FUNCTION_BLOCK CMD_bloc (* Basic Function Block Type *)
  (* Standard: 61499-2 *)
  (* Version 0.0, 13/06/2022, Etienne, Schneider Electric, Template *)
  PACKAGE Main;
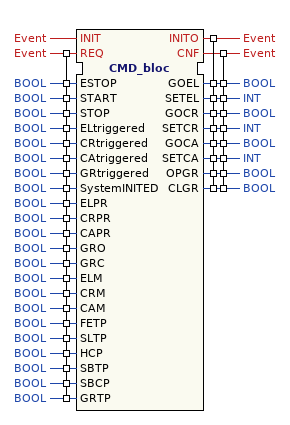
  EVENT_INPUT
    INIT; (* Initialization Request *)
    REQ WITH ESTOP, START, STOP, ELtriggered, CRtriggered, CAtriggered, GRtriggered, SystemINITED, ELPR, CRPR, CAPR, GRO, GRC, ELM, CRM, CAM, HCP, SBTP, SBCP, FETP, SLTP, GRTP; (* Normal Execution Request *)
  END_EVENT
  EVENT_OUTPUT
    INITO WITH GOEL, SETEL, GOCA, SETCA, GOCR, SETCR, OPGR, CLGR; (* Initialization Confirm *)
    CNF WITH GOEL, SETEL, GOCA, SETCA, GOCR, SETCR, OPGR, CLGR; (* Execution Confirmation *)
  END_EVENT
  VAR_INPUT
    ESTOP : BOOL;
    START : BOOL;
    STOP : BOOL;
    ELtriggered : BOOL;
    CRtriggered : BOOL;
    CAtriggered : BOOL;
    GRtriggered : BOOL;
    SystemINITED : BOOL;
    ELPR : BOOL;
    CRPR : BOOL;
    CAPR : BOOL;
    GRO : BOOL;
    GRC : BOOL;
    ELM : BOOL;
    CRM : BOOL;
    CAM : BOOL;
    FETP : BOOL;
    SLTP : BOOL;
    HCP : BOOL;
    SBTP : BOOL;
    SBCP : BOOL;
    GRTP : BOOL;
  END_VAR
  VAR_OUTPUT
    GOEL : BOOL; (* Output event qualifier *)
    SETEL : INT;
    GOCR : BOOL;
    SETCR : INT;
    GOCA : BOOL;
    SETCA : INT;
    OPGR : BOOL;
    CLGR : BOOL;
  END_VAR
  VAR
    i : INT;
  END_VAR
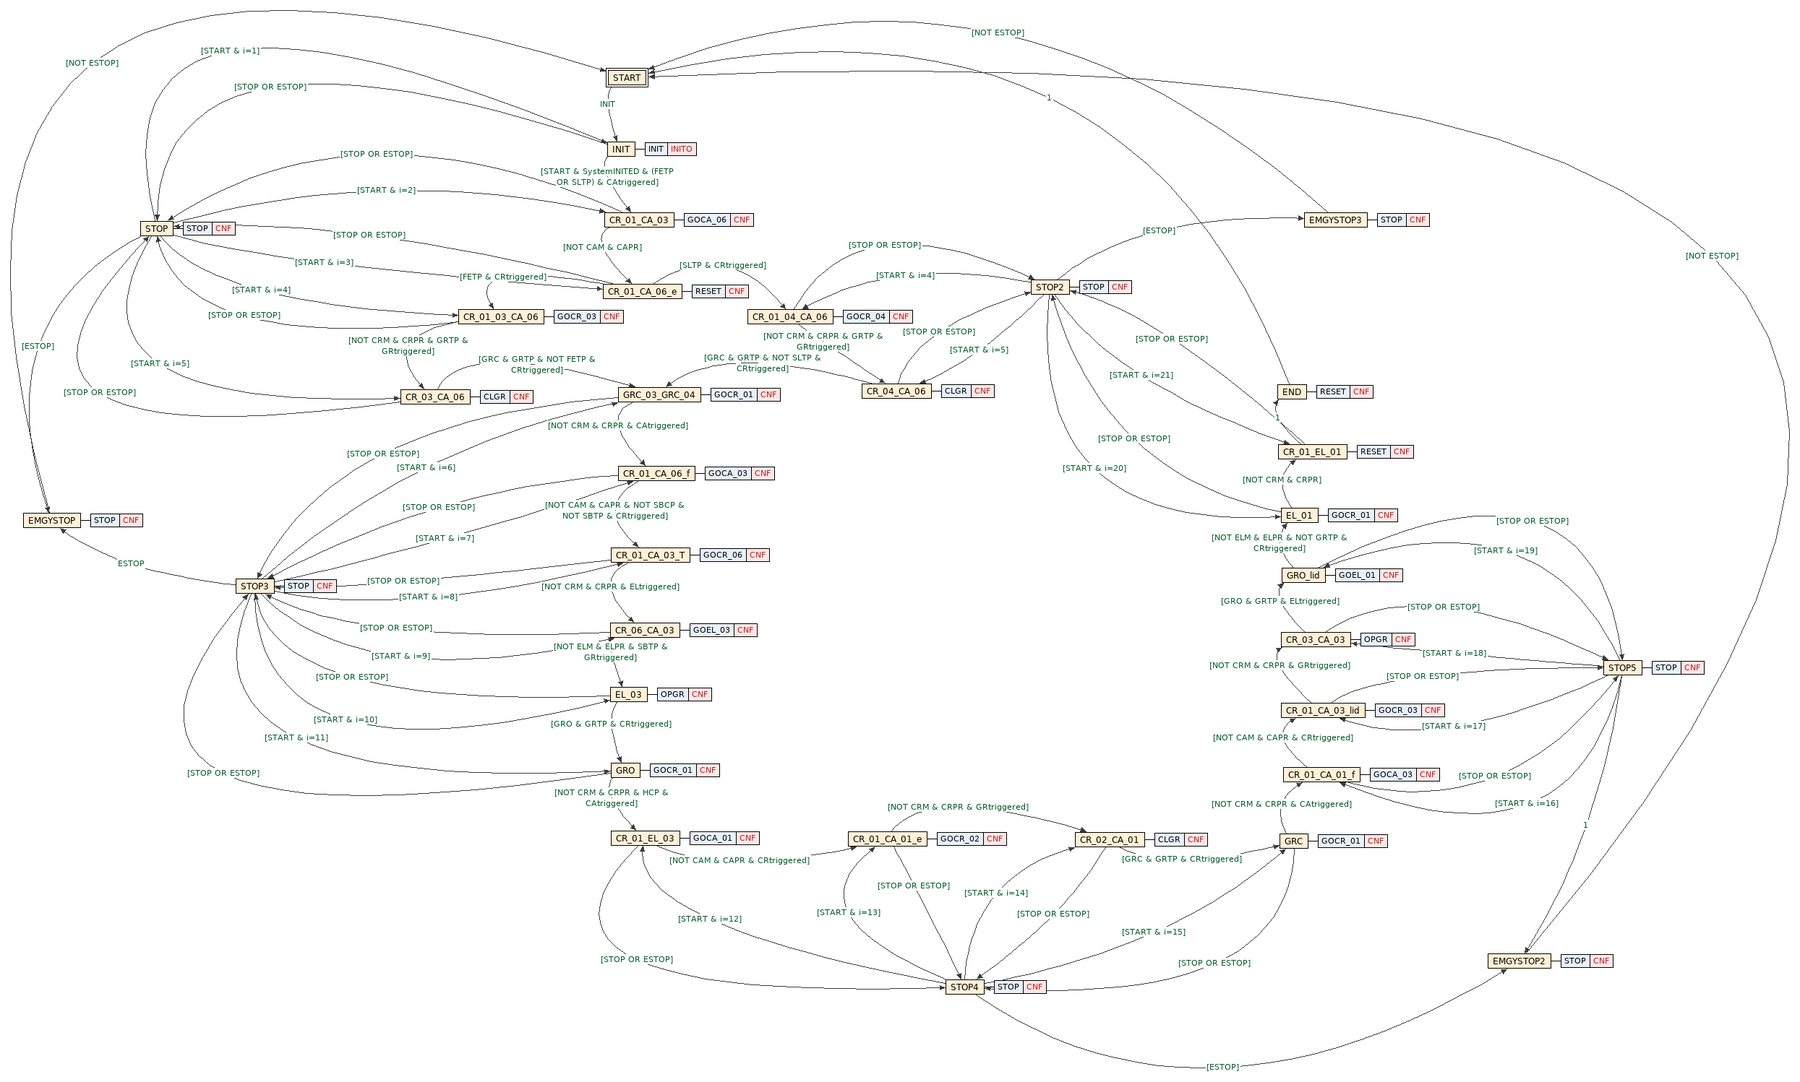
  EC_STATES
    START; (* Initial State *)
    INIT : INIT -> INITO; (* Initialization *)
    CR_01_CA_03 : GOCA_06 -> CNF;
    CR_01_03_CA_06 : GOCR_03 -> CNF;
    CR_01_04_CA_06 : GOCR_04 -> CNF;
    GRC_03_GRC_04 : GOCR_01 -> CNF;
    CR_01_CA_06_f : GOCA_03 -> CNF;
    CR_01_CA_03_T : GOCR_06 -> CNF;
    CR_06_CA_03 : GOEL_03 -> CNF;
    EL_03 : OPGR -> CNF;
    GRO : GOCR_01 -> CNF;
    EL_01 : GOCR_01 -> CNF;
    CR_01_EL_03 : GOCA_01 -> CNF;
    END : RESET -> CNF;
    CR_01_CA_01_e : GOCR_02 -> CNF;
    CR_02_CA_01 : CLGR -> CNF;
    GRC : GOCR_01 -> CNF;
    CR_01_CA_01_f : GOCA_03 -> CNF;
    CR_01_CA_03_lid : GOCR_03 -> CNF;
    CR_03_CA_03 : OPGR -> CNF;
    GRO_lid : GOEL_01 -> CNF;
    CR_01_EL_01 : RESET -> CNF;
    CR_01_CA_06_e : RESET -> CNF;
    CR_03_CA_06 : CLGR -> CNF;
    CR_04_CA_06 : CLGR -> CNF;
    STOP : STOP -> CNF;
    STOP2 : STOP -> CNF;
    STOP3 : STOP -> CNF;
    STOP4 : STOP -> CNF;
    STOP5 : STOP -> CNF;
    EMGYSTOP : STOP -> CNF;
    EMGYSTOP2 : STOP -> CNF;
    EMGYSTOP3 : STOP -> CNF;
  END_STATES
  EC_TRANSITIONS
    START TO INIT := INIT;
    CR_01_03_CA_06 TO CR_03_CA_06 := [NOT CRM & CRPR & GRTP & GRtriggered];
    CR_01_04_CA_06 TO CR_04_CA_06 := [NOT CRM & CRPR & GRTP & GRtriggered];
    GRC_03_GRC_04 TO CR_01_CA_06_f := [NOT CRM & CRPR & CAtriggered];
    CR_01_CA_06_f TO CR_01_CA_03_T := [NOT CAM & CAPR & NOT SBCP & NOT SBTP & CRtriggered];
    CR_01_CA_03_T TO CR_06_CA_03 := [NOT CRM & CRPR & ELtriggered];
    CR_06_CA_03 TO EL_03 := [NOT ELM & ELPR & SBTP & GRtriggered];
    EL_03 TO GRO := [GRO & GRTP & CRtriggered];
    GRO TO CR_01_EL_03 := [NOT CRM & CRPR & HCP & CAtriggered];
    CR_01_EL_03 TO CR_01_CA_01_e := [NOT CAM & CAPR & CRtriggered];
    CR_01_CA_01_e TO CR_02_CA_01 := [NOT CRM & CRPR & GRtriggered];
    CR_02_CA_01 TO GRC := [GRC & GRTP & CRtriggered];
    GRC TO CR_01_CA_01_f := [NOT CRM & CRPR & CAtriggered];
    CR_01_CA_01_f TO CR_01_CA_03_lid := [NOT CAM & CAPR & CRtriggered];
    CR_01_CA_03_lid TO CR_03_CA_03 := [NOT CRM & CRPR & GRtriggered];
    CR_03_CA_03 TO GRO_lid := [GRO & GRTP & ELtriggered];
    GRO_lid TO EL_01 := [NOT ELM & ELPR & NOT GRTP & CRtriggered];
    EL_01 TO CR_01_EL_01 := [NOT CRM & CRPR];
    END TO START := 1;
    CR_01_CA_03 TO CR_01_CA_06_e := [NOT CAM & CAPR];
    CR_01_CA_06_e TO CR_01_03_CA_06 := [FETP & CRtriggered];
    CR_01_CA_06_e TO CR_01_04_CA_06 := [SLTP & CRtriggered];
    CR_03_CA_06 TO GRC_03_GRC_04 := [GRC & GRTP & NOT FETP & CRtriggered];
    CR_04_CA_06 TO GRC_03_GRC_04 := [GRC & GRTP & NOT SLTP & CRtriggered];
    INIT TO STOP := [STOP OR ESTOP];
    CR_01_CA_03 TO STOP := [STOP OR ESTOP];
    CR_01_CA_06_e TO STOP := [STOP OR ESTOP];
    CR_01_03_CA_06 TO STOP := [STOP OR ESTOP];
    CR_03_CA_06 TO STOP := [STOP OR ESTOP];
    CR_01_04_CA_06 TO STOP2 := [STOP OR ESTOP];
    CR_04_CA_06 TO STOP2 := [STOP OR ESTOP];
    EL_01 TO STOP2 := [STOP OR ESTOP];
    CR_01_EL_01 TO STOP2 := [STOP OR ESTOP];
    GRC_03_GRC_04 TO STOP3 := [STOP OR ESTOP];
    CR_01_CA_06_f TO STOP3 := [STOP OR ESTOP];
    CR_01_CA_03_T TO STOP3 := [STOP OR ESTOP];
    CR_06_CA_03 TO STOP3 := [STOP OR ESTOP];
    EL_03 TO STOP3 := [STOP OR ESTOP];
    GRO TO STOP3 := [STOP OR ESTOP];
    CR_01_EL_03 TO STOP4 := [STOP OR ESTOP];
    CR_01_CA_01_e TO STOP4 := [STOP OR ESTOP];
    CR_02_CA_01 TO STOP4 := [STOP OR ESTOP];
    GRC TO STOP4 := [STOP OR ESTOP];
    CR_01_CA_01_f TO STOP5 := [STOP OR ESTOP];
    CR_01_CA_03_lid TO STOP5 := [STOP OR ESTOP];
    CR_03_CA_03 TO STOP5 := [STOP OR ESTOP];
    GRO_lid TO STOP5 := [STOP OR ESTOP];
    STOP TO INIT := [START & i=1];
    STOP TO CR_01_03_CA_06 := [START & i=4];
    STOP TO CR_03_CA_06 := [START & i=5];
    STOP TO CR_01_CA_06_e := [START & i=3];
    STOP TO CR_01_CA_03 := [START & i=2];
    STOP3 TO GRC_03_GRC_04 := [START & i=6];
    STOP3 TO CR_01_CA_06_f := [START & i=7];
    STOP3 TO CR_01_CA_03_T := [START & i=8];
    STOP3 TO CR_06_CA_03 := [START & i=9];
    STOP3 TO EL_03 := [START & i=10];
    STOP3 TO GRO := [START & i=11];
    STOP4 TO CR_01_EL_03 := [START & i=12];
    STOP4 TO CR_01_CA_01_e := [START & i=13];
    STOP4 TO CR_02_CA_01 := [START & i=14];
    STOP4 TO GRC := [START & i=15];
    STOP5 TO CR_01_CA_01_f := [START & i=16];
    STOP5 TO CR_01_CA_03_lid := [START & i=17];
    STOP5 TO CR_03_CA_03 := [START & i=18];
    STOP5 TO GRO_lid := [START & i=19];
    STOP2 TO CR_01_04_CA_06 := [START & i=4];
    STOP2 TO CR_04_CA_06 := [START & i=5];
    STOP2 TO CR_01_EL_01 := [START & i=21];
    STOP2 TO EL_01 := [START & i=20];
    STOP3 TO EMGYSTOP := ESTOP;
    STOP TO EMGYSTOP := [ESTOP];
    EMGYSTOP TO START := [NOT ESTOP];
    STOP4 TO EMGYSTOP2 := [ESTOP];
    STOP5 TO EMGYSTOP2 := 1;
    STOP2 TO EMGYSTOP3 := [ESTOP];
    EMGYSTOP3 TO START := [NOT ESTOP];
    EMGYSTOP2 TO START := [NOT ESTOP];
    INIT TO CR_01_CA_03 := [START & SystemINITED & (FETP OR SLTP) & CAtriggered];
    CR_01_EL_01 TO END := 1;
  END_TRANSITIONS
  ALGORITHM INIT IN ST: (* Initialization algorithm *)
;
i:=1;
  END_ALGORITHM
  ALGORITHM GOCA_06 IN ST:
;
GOCA := TRUE;
SETCA := 1320;
i:=i+1;

GOEL := FALSE;
GOCR := FALSE;
  END_ALGORITHM
  ALGORITHM GOCR_03 IN ST:
;
GOCR := TRUE;
SETCR := 54;

GOCA := FALSE;
GOEL := FALSE;

i:=i+1;
  END_ALGORITHM
  ALGORITHM GOCR_04 IN ST:
;
GOCR := TRUE;
SETCR := 81;

GOEL := FALSE;
GOCA := FALSE;

i:=i+1;
  END_ALGORITHM
  ALGORITHM CLGR IN ST:
;
CLGR := TRUE;
OPGR := FALSE;

GOCR := FALSE;
GOEL := FALSE;
GOCA := FALSE;

i:=i+1;
  END_ALGORITHM
  ALGORITHM GOCR_01 IN ST:
;
GOCR := TRUE;
SETCR := -2;

GOCA := FALSE;
GOEL := FALSE;

FETP := FALSE;
SLTP := FALSE;

i:=i+1;
  END_ALGORITHM
  ALGORITHM GOCA_03 IN ST:
;
GOCA := TRUE;
SETCA := 538;

GOEL := FALSE;
GOCR := FALSE;

i:=i+1;
  END_ALGORITHM
  ALGORITHM GOCR_06 IN ST:
;
GOCR := TRUE;
SETCR := 261;

GOCA := FALSE;
GOEL := FALSE;

i:=i+1;
  END_ALGORITHM
  ALGORITHM GOEL_03 IN ST:
;
GOEL := TRUE;
SETEL := 274;

GOCA := FALSE;
GOCR := FALSE;

i:=i+1;
  END_ALGORITHM
  ALGORITHM OPGR IN ST:
;
CLGR := FALSE;
OPGR := TRUE;

GOCR := FALSE;
GOEL := FALSE;
GOCA := FALSE;

i:=i+1;
  END_ALGORITHM
  ALGORITHM GOCA_01 IN ST:
;
GOCA := TRUE;
SETCA := 10;

GOEL := FALSE;
GOCR := FALSE;

i:=i+1;
  END_ALGORITHM
  ALGORITHM GOCR_02 IN ST:
;
GOCR := TRUE;
SETCR := 41;

GOCA := FALSE;
GOEL := FALSE;

i:=i+1;
  END_ALGORITHM
  ALGORITHM GOCR_XX IN ST:
;
GOCR := TRUE;
SETCR := 00;

GOCA := FALSE;
GOEL := FALSE;
  END_ALGORITHM
  ALGORITHM GOEL_01 IN ST:
;
GOEL := TRUE;
SETEL := -2;

GOCA := FALSE;
GOCR := FALSE;

i:=i+1;
  END_ALGORITHM
  ALGORITHM RESET IN ST:
;
GOCA := FALSE;
GOCR := FALSE;
GOEL := FALSE;
OPGR := FALSE;
CLGR := FALSE;

i:=i+1;
  END_ALGORITHM
  ALGORITHM STOP IN ST:
;
GOCA := FALSE;
GOCR := FALSE;
GOEL := FALSE;
OPGR := FALSE;
CLGR := FALSE;
  END_ALGORITHM
END_FUNCTION_BLOCK
